{attribute 'pack_mode':='1'}
TYPE PerturbToteParams :
STRUCT
   target_id: ModelIdentifier;
END_STRUCT
END_TYPE

(* stored: Version 1.1.0.1, ProductVersion 3.1.4024.12
   DUT PerturbToteParams: Id {97f7dfca-1c3c-41d1-8410-ca45f5cadf78} *)
